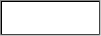
VISUALIZATION VISU_HMI_SUBSUBSYSTEM_BUTTON  // 101x36
VAR_IN_OUT
    m_Hmi : FB_HMI_BUTTON;
END_VAR
    Rectangle (0,0 100x35), invisible if: m_Hmi.bIsNotOrange
    Rectangle (0,0 100x35), invisible if: m_Hmi.bIsNotGray
    Rectangle (0,0 100x35), invisible if: m_Hmi.bIsNotBlue
    Rectangle (0,0 100x35), invisible if: m_Hmi.bIsNotRed
    Rectangle (0,0 100x35), invisible if: m_Hmi.bIsNotGreen
    Rectangle (0,0 100x35), "%s", text variable: m_Hmi.sName
    Rectangle (0,0 100x35), invisible if: m_Hmi.bNotActivated
    Line (0,34) (100,34), invisible if: m_Hmi.bActivated
    Line (99,0) (99,35), invisible if: m_Hmi.bActivated
    Line (98,0) (0,0), invisible if: m_Hmi.bActivated
    Line (0,35) (0,0), invisible if: m_Hmi.bActivated
    Line (100,35) (100,1), invisible if: m_Hmi.bNotActivated
    Line (0,1) (99,1), invisible if: m_Hmi.bNotActivated
    Line (1,0) (1,35), invisible if: m_Hmi.bNotActivated
    Line (100,35) (1,35), invisible if: m_Hmi.bNotActivated
END_VISUALIZATION

(* stored: Version 1.1.0.1, ProductVersion 3.1.4024.14
   Visu VISU_HMI_SUBSUBSYSTEM_BUTTON: Id {202beae4-be49-4542-a734-b3ea423bf0f8} *)
